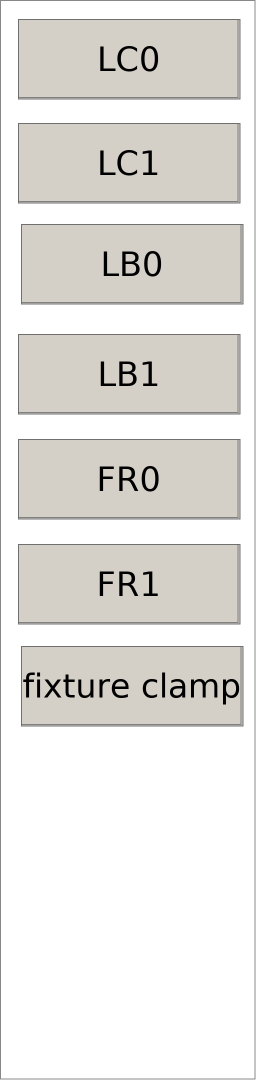
VISUALIZATION OtherList  // 256x1080
    Button (18,19 222x80), "LC0", colour toggle: G_HMI.iOthers =0
        p573394764: 16#FF00FF00
        OnMouseDown: execute {
            G_HMI.iLc  := 0;
            G_HMI.iMainFrame	:= 2;
            G_HMI.iOthers	:= 0;
        }
    Button (21,224 222x80), "LB0", colour toggle: G_HMI.iOthers =2
        p573394764: 16#FF00FF00
        OnMouseDown: execute {
            G_HMI.iLb  := 0;
            G_HMI.iMainFrame	:= 3;
            G_HMI.iOthers	:= 2;
        }
    Button (18,123 222x80), "LC1", colour toggle: G_HMI.iOthers =1
        p573394764: 16#FF00FF00
        OnMouseDown: execute {
            G_HMI.iLc  := 1;
            G_HMI.iMainFrame	:= 2;
            G_HMI.iOthers	:= 1;
        }
    Button (18,334 222x80), "LB1", colour toggle: G_HMI.iOthers =3
        p573394764: 16#FF00FF00
        OnMouseDown: execute {
            G_HMI.iLb  := 1;
            G_HMI.iMainFrame	:= 3;
            G_HMI.iOthers	:= 3;
        }
    Button (18,439 222x80), "FR0", colour toggle: G_HMI.iOthers =4
        p573394764: 16#FF00FF00
        OnMouseDown: execute {
            G_HMI.iFr  := 0;
            G_HMI.iMainFrame	:= 4;
            G_HMI.iOthers	:= 4;
        }
    Button (18,544 222x80), "FR1", colour toggle: G_HMI.iOthers =5
        p573394764: 16#FF00FF00
        OnMouseDown: execute {
            G_HMI.iFr  := 1;
            G_HMI.iMainFrame	:= 4;
            G_HMI.iOthers	:= 5;
        }
    Button (21,646 222x80), "fixture clamp", colour toggle: G_HMI.iOthers =6
        p573394764: 16#FF00FF00
        OnMouseDown: execute { G_HMI.iMainFrame	:= 5; G_HMI.iOthers	:= 6; }
END_VISUALIZATION

(* stored: Version 1.1.0.1, ProductVersion 3.1.4024.12
   Visu OtherList: Id {c6646ba3-95c6-4885-9a92-385fe668c684} *)
